FUNCTION_BLOCK PUBLIC FB_RtrigFtrig
VAR_INPUT
	bIn : BOOL;
END_VAR
VAR_OUTPUT
	// rising trigger bIn
	bRq : BOOL;
	// falling trigger bIn
	bFq : BOOL;
END_VAR
VAR
	rtrig : R_TRIG;
	ftrig : F_TRIG;
END_VAR

rtrig(CLK := bIn, Q => bRq);
ftrig(CLK := bIn, Q => bFq);

END_FUNCTION_BLOCK

(* stored: Version 1.1.0.1
   POU FB_RtrigFtrig: Id {2cd37571-fd4a-4532-bf6a-19e4578ef0be}, SpecialFunc None *)
